// Mitsubishi GX Works2 project: 0702fullver   PLC: Q03UDV

// global labels: Global1
VAR_GLOBAL
  공급후진리드 AT X20 : BOOL;
  공급전진리드 AT X21 : BOOL;
  매거진센서 AT X22 : BOOL;
  고주파센서 AT X23 : BOOL;
  용량형센서 AT X24 : BOOL;
  근접포토센서 AT X25 : BOOL;
  그리퍼온리드 AT X27 : BOOL;
  그리퍼오프리드 AT X28 : BOOL;
  물품도착포토 AT X29 : BOOL;
  TG1 AT X2A : BOOL;
  TG2 AT X2B : BOOL;
  TG3 AT X2C : BOOL;
  PB4 AT X2D : BOOL;
  PB5 AT X2E : BOOL;
  창고1 AT X30 : BOOL;
  창고2 AT X31 : BOOL;
  창고3 AT X32 : BOOL;
  창고4 AT X33 : BOOL;
  창고5 AT X34 : BOOL;
  창고6 AT X35 : BOOL;
  창고7 AT X36 : BOOL;
  창고8 AT X37 : BOOL;
  창고9 AT X38 : BOOL;
  도어센서 AT X39 : BOOL;
  압력센서 AT X3A : BOOL;
  공급전솔 AT Y40 : BOOL;
  공급후솔 AT Y41 : BOOL;
  그리퍼온솔 AT Y42 : BOOL;
  그리퍼오프솔 AT Y43 : BOOL;
  경광녹색 AT Y44 : BOOL;
  경광황색 AT Y45 : BOOL;
  경광적색 AT Y46 : BOOL;
  부저 AT Y47 : BOOL;
  컨베이어 AT Y48 : BOOL;
  램프1 AT Y4A : BOOL;
  램프2 AT Y4B : BOOL;
  램프3 AT Y4C : BOOL;
  램프5 AT Y4D : BOOL;
  램프4 AT Y4E : BOOL;
  R그립온명령 AT X1000 : BOOL;
  R그립오프명령 AT X1001 : BOOL;
  R_PLC시작 AT X1002 : BOOL;
  R_판별리셋 AT X1003 : BOOL;
  R재공급 AT X1004 : BOOL;
  R그립온센서 AT Y1000 : BOOL;
  R그립오프센서 AT Y1001 : BOOL;
  R물품없음 AT Y1002 : BOOL;
  R_금속 AT Y1003 : BOOL;
  R_검비금속 AT Y1004 : BOOL;
  R_흰비금속 AT Y1005 : BOOL;
  R물품도착 AT Y1006 : BOOL;
  R컨베이어 AT Y1007 : BOOL;
  R_재시작 AT Y1008 : BOOL;
  R_interrupt AT Y1009 : BOOL;
  R창고1 AT Y100A : BOOL;
  R창고2 AT Y100B : BOOL;
  R창고3 AT Y100C : BOOL;
  R창고4 AT Y100D : BOOL;
  R창고5 AT Y100E : BOOL;
  R창고6 AT Y100F : BOOL;
  R창고7 AT Y1010 : BOOL;
  R창고8 AT Y1011 : BOOL;
  R창고9 AT Y1012 : BOOL;
  R창고A AT Y1013 : BOOL;
END_VAR

PROGRAM MAIN
VAR
  PLC공정중 : BOOL;
  공급전진 : BOOL;
  공급후진 : BOOL;
  용량형탐지 : BOOL;
  고주파탐지 : BOOL;
  근접포토탐지 : BOOL;
  T_도착지연 : TIMER;
  T_매거진지연 : TIMER;
  컨구동 : BOOL;
  컨정지 : BOOL;
  금속 : BOOL;
  흰플 : BOOL;
  블플 : BOOL;
  T_판별지연 : TIMER;
  검플 : BOOL;
  물품도착 : BOOL;
  T_공정지연 : TIMER;
  공정종료 : BOOL;
END_VAR
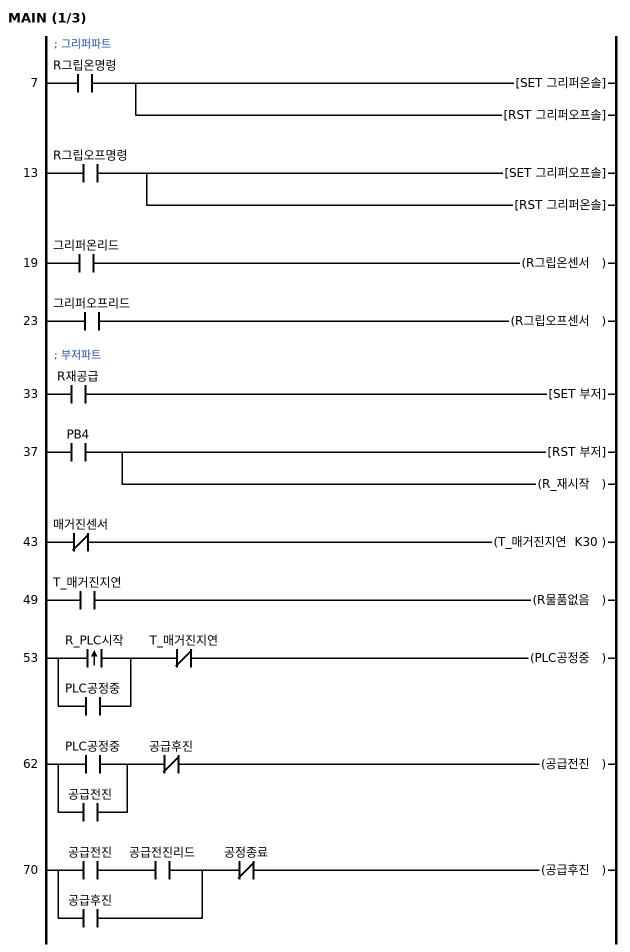
; 그리퍼파트
7     LD      R그립온명령
      SET     그리퍼온솔
      RST     그리퍼오프솔
13    LD      R그립오프명령
      SET     그리퍼오프솔
      RST     그리퍼온솔
19    LD      그리퍼온리드
      OUT     R그립온센서
23    LD      그리퍼오프리드
      OUT     R그립오프센서
; 부저파트
33    LD      R재공급
      SET     부저
37    LD      PB4
      RST     부저
      OUT     R_재시작
43    LDI     매거진센서
      OUT     T_매거진지연 K30
49    LD      T_매거진지연
      OUT     R물품없음
53    LDP     R_PLC시작
      OR      PLC공정중
      ANI     T_매거진지연
      OUT     PLC공정중
62    LD      PLC공정중
      OR      공급전진
      ANI     공급후진
      OUT     공급전진
70    LD      공급전진
      AND     공급전진리드
      OR      공급후진
      ANI     공정종료
      OUT     공급후진
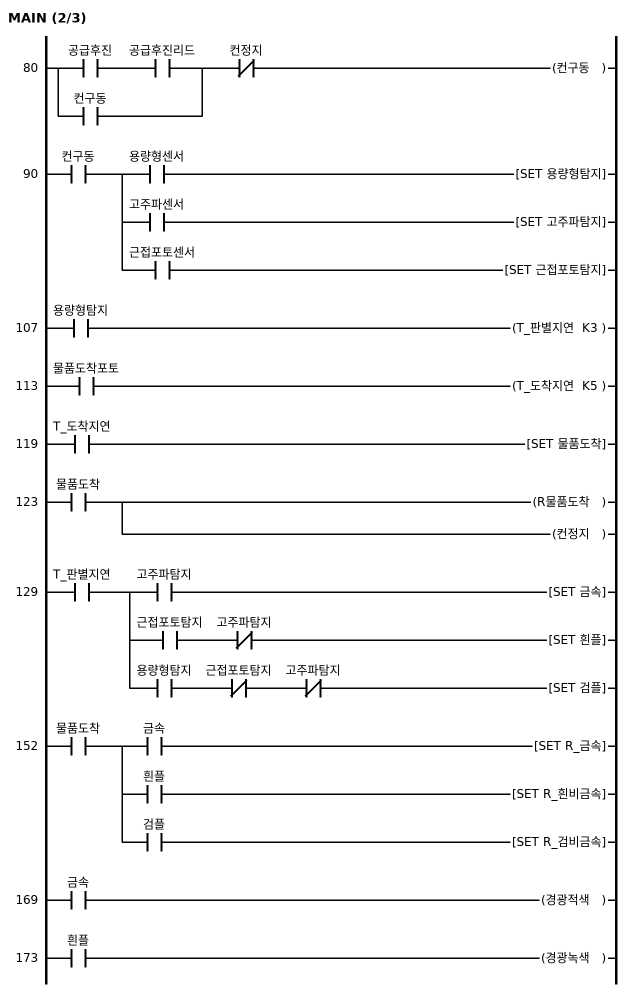
80    LD      공급후진
      AND     공급후진리드
      OR      컨구동
      ANI     컨정지
      OUT     컨구동
90    LD      컨구동
      MPS
      AND     용량형센서
      SET     용량형탐지
      MRD
      AND     고주파센서
      SET     고주파탐지
      MPP
      AND     근접포토센서
      SET     근접포토탐지
107   LD      용량형탐지
      OUT     T_판별지연 K3
113   LD      물품도착포토
      OUT     T_도착지연 K5
119   LD      T_도착지연
      SET     물품도착
123   LD      물품도착
      OUT     R물품도착
      OUT     컨정지
129   LD      T_판별지연
      MPS
      AND     고주파탐지
      SET     금속
      MRD
      AND     근접포토탐지
      ANI     고주파탐지
      SET     흰플
      MPP
      AND     용량형탐지
      ANI     근접포토탐지
      ANI     고주파탐지
      SET     검플
152   LD      물품도착
      MPS
      AND     금속
      SET     R_금속
      MRD
      AND     흰플
      SET     R_흰비금속
      MPP
      AND     검플
      SET     R_검비금속
169   LD      금속
      OUT     경광적색
173   LD      흰플
      OUT     경광녹색
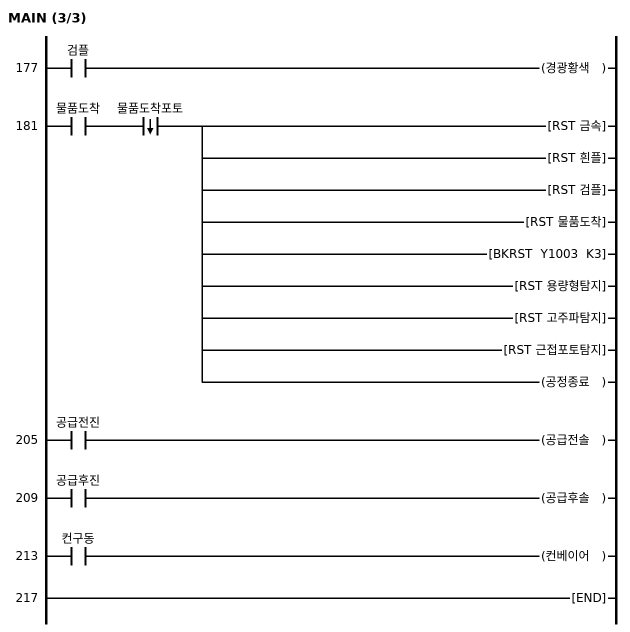
177   LD      검플
      OUT     경광황색
181   LD      물품도착
      ANDF    물품도착포토
      RST     금속
      RST     흰플
      RST     검플
      RST     물품도착
      BKRST   Y1003 K3
      RST     용량형탐지
      RST     고주파탐지
      RST     근접포토탐지
      OUT     공정종료
205   LD      공급전진
      OUT     공급전솔
209   LD      공급후진
      OUT     공급후솔
213   LD      컨구동
      OUT     컨베이어
217   END
END_PROGRAM
